{attribute 'qualified_only'}
//{attribute 'strict'}
TYPE SectionTask :
(
	IDLE,
	ALIGN,
	ACTIVE,
	DISCHARGE,
	COMPLETE,
	
	size
);
END_TYPE

(* stored: Version 1.1.0.1, ProductVersion 3.1.4024.11
   DUT SectionTask: Id {9750fdd6-c9e6-4c18-b005-35290999abad} *)
